INTERFACE I_SimpleLogArgument EXTENDS I_Base,I_ToString

END_INTERFACE

(* stored: Version 1.1.0.1
   Itf I_SimpleLogArgument: Id {6728e269-28d4-4a66-819c-dae3f5d4d360} *)
